VAR_GLOBAL
	INIT_Execute1 : BOOL;
	INIT_Execute2 : BOOL;
	INIT_Execute3 : BOOL;
	INIT_Execute4 : BOOL;
	INIT_Execute5 : BOOL;
	INIT_Execute6 : BOOL;
END_VAR

(* stored: Version 1.1.0.1, ProductVersion 3.1.4024.0
   GVL INIT_GVL: Id {eb7b0bf5-2e7f-4ee9-9725-974a11e67728} *)
